FUNCTION_BLOCK FB_QuantityINTPublicMock EXTENDS FB_FalliblePublicMock IMPLEMENTS I_QuantityINT
VAR
    nVal : INT;
    sUnits : T_MaxString;
END_VAR


METHOD Copy
VAR_INPUT
    QuantityToCopy : I_QuantityINT;
END_VAR

Val := QuantityToCopy.Val;
Units := QuantityToCopy.Units;

IF QuantityToCopy.GetError() THEN
    SetError(Msg := QuantityToCopy.GetErrorMsg());
ELSE
    ClearError();
END_IF
END_METHOD


METHOD Equals : BOOL
VAR_INPUT
    Quantity	: I_QuantityINT;
END_VAR

Equals := Quantity.Units = Units AND Quantity.Val = Val;
END_METHOD


PROPERTY Units : T_MaxString
GET

Units := sUnits;
END_GET
SET

sUnits := Units;
END_SET
END_PROPERTY


PROPERTY Val : INT
GET

Val := THIS^.nVal;
END_GET
SET

THIS^.nVal := Val;
END_SET
END_PROPERTY

END_FUNCTION_BLOCK

(* stored: Version 1.1.0.1
   POU FB_QuantityINTPublicMock: Id {25a1d111-4045-47b7-859c-1db48ea9bedf}, SpecialFunc None
   Method Copy: Id {2750d99e-b0cb-4ae8-85e0-f3708d488206}
   Method Equals: Id {1947b1d1-c2a2-456d-afe6-cdf6e06bcaf0}
   Property Units: Id {04680986-f99a-4221-a383-34b986d809d4}
   Get Get: Id {ff38750f-3172-428e-96a8-893ff8478e42}
   Set Set: Id {278d3eed-2b0b-448c-957c-67a2427ee7ac}
   Property Val: Id {1388d4ff-d7bf-4c33-ae6d-7a137c96929d}
   Get Get: Id {e281da4e-4dc4-4aca-801f-3155e3fabfe6}
   Set Set: Id {f1c02087-ad76-4076-8c49-3337df0388b7} *)
